{attribute 'GeneratedUsingTerminal: EL3403-0000-0023'}
{attribute addProperty BoxType "EL3403-0000-0023"}
{attribute addProperty Id "IndexAT %Q*USINT1"}
{attribute addProperty CRC "3858488880"}
{attribute addProperty Size "1"}
TYPE PM_Outputs_Channel_E5FBDE30 EXTENDS TcoIo.OutputBase_10CEE7DE :
STRUCT
	{attribute addProperty Name "Index"}
	Index AT %Q* : USINT;
END_STRUCT
END_TYPE

(* stored: Version 1.2.0.0, ProductVersion 3.1.4024.9
   DUT PM_Outputs_Channel_E5FBDE30: Id {fbf5e09c-5a39-0baa-155b-1f1894b059eb} *)
